{attribute 'GeneratedUsingTerminal: EL2911-0000-0016'}
{attribute addProperty BoxType "EL2911-0000-0016"}
{attribute addProperty Id "FSOEAT %Q*FSOE_EE2DB9C38"}
{attribute addProperty CRC "4147897402"}
{attribute addProperty Size "8"}
TYPE FSoE_Outputs_F73BE43A EXTENDS OutputBase_10CEE7DE :
STRUCT
	{attribute addProperty Name "FSOE"}
	FSOE AT %Q* : FSOE_EE2DB9C3;
END_STRUCT
END_TYPE

(* stored: Version 1.2.0.0, ProductVersion 3.1.4024.9
   DUT FSoE_Outputs_F73BE43A: Id {437a3c63-973e-4961-b776-517c864d80b5} *)
